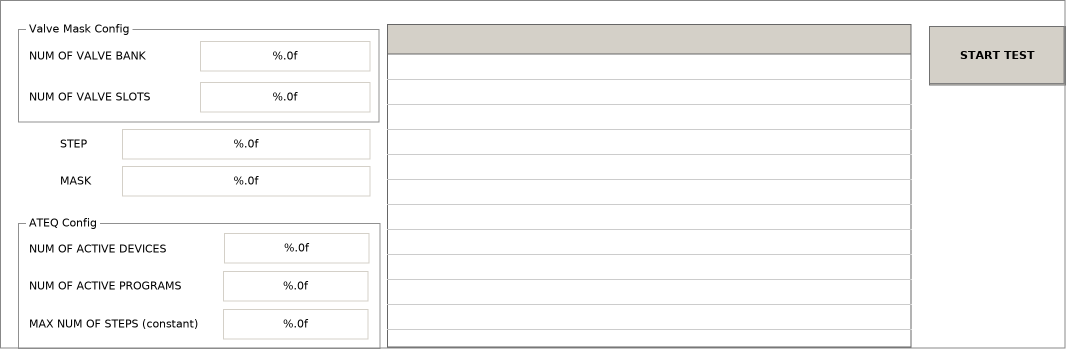
VISUALIZATION visuMain  // 1066x349
    Table (387,24 524x323), data array: GVL_TcHmi.anValveMaskListToDisplay
        p3854506369: GVL_TcHmi.anValveMaskListToDisplay[INDEX]
        p2232123230: GVL_VisuControlHMI.anValveMaskListToDisplay[INDEX]
    Textfield (122,129 248x30), "%.0f", text variable: GVL_TcHmi.visValveMaskIdx
        OnMouseClick: write GVL_TcHmi.visValveMaskIdx via VisuDialogs.Numpad
    Label (57,129 60x30), "STEP"
    Textfield (122,129 248x30), "%.0f", text variable: GVL_TcHmi.visValveMaskIdx
        OnMouseClick: write GVL_TcHmi.visValveMaskIdx via VisuDialogs.Numpad
    Textfield (122,129 248x30), "%.0f", text variable: GVL_TcHmi.visValveMaskIdx
        OnMouseClick: write GVL_TcHmi.visValveMaskIdx via VisuDialogs.Numpad
    Textfield (122,129 248x30), "%.0f", text variable: GVL_TcHmi.visValveMaskIdx
        OnMouseClick: write GVL_TcHmi.visValveMaskIdx via Default, min 0, max nNumOfActiveProgramsToRun
    Textfield (122,166 248x30), "%.0f", text variable: GVL_TcHmi.nValveMask
        OnMouseClick: write GVL_TcHmi.nValveMask via VisuDialogs.Numpad
    Label (57,166 60x30), "MASK"
    Textfield (122,166 248x30), "%.0f", text variable: GVL_TcHmi.nValveMask
        OnMouseClick: write GVL_TcHmi.nValveMask via VisuDialogs.Numpad
    Textfield (122,166 248x30), "%.0f", text variable: GVL_TcHmi.nValveMask
        OnMouseClick: write GVL_TcHmi.nValveMask via VisuDialogs.Numpad
    Textfield (122,166 248x30), "%.0f", text variable: GVL_TcHmi.nValveMask
        OnMouseClick: write GVL_TcHmi.nValveMask via Default
    GroupBox (18,21 361x101), "Valve Mask Config"
    Label (26,234 182x30), "NUM OF ACTIVE DEVICES"
    Textfield (223,271 145x30), "%.0f", text variable: nNumOfActiveProgramsToRun
        OnMouseClick: write nNumOfActiveProgramsToRun via Default, format %.0f
    Label (26,271 182x30), "NUM OF ACTIVE PROGRAMS"
    Textfield (223,309 145x30), "%.0f", text variable: nMaxTestCount
        OnMouseClick: write nMaxTestCount via Default, format %.0f
    Label (26,309 182x30), "MAX NUM OF STEPS (constant)"
    GroupBox (18,215 362x134), "ATEQ Config"
    Label (26,41 141x30), "NUM OF VALVE BANK"
    Textfield (200,82 170x30), "%.0f", text variable: nMaxNumOfValveSlots
        OnMouseClick: write nMaxNumOfValveSlots via VisuDialogs.Numpad
    Label (26,82 141x30), "NUM OF VALVE SLOTS"
    Textfield (224,233 145x30), "%.0f", text variable: GVL_AteqConfig.nNumOfActiveDevices
        OnMouseClick: write GVL_AteqConfig.nNumOfActiveDevices via Default, format %.0f
    Textfield (200,41 170x30), "%.0f", text variable: nActiveValveBanks
        OnMouseClick: write nActiveValveBanks via Default, format %.0f
    Button (929,26 137x59), "START TEST"
        OnMouseClick: toggle GVL_AteqConfig.abAutoTestRecipeStart
END_VISUALIZATION

(* stored: Version 1.1.0.1
   Visu visuMain: Id {13b731d7-6b83-043b-0600-952922f53888} *)
